// TIA Portal V20 export
DATA_BLOCK "G"   // DB350
{ S7_Optimized_Access := 'TRUE' }
// stored: AutoNumber false, IsRetainMemResEnabled true, MemoryReserve 100, RetainMemoryReserve 100
   VAR RETAIN
      lampTest : Bool;   // lamp test
      settingMode : Bool;   // setting mode active
      jogMode : Bool;   // jog mode active
      scannerReady : Bool;   // scanner ready
      scannerErr : Bool;   // scanner error
      scannerEmpty : Bool;   // scanner empty
      releaseInfeed : Bool;   // release infeed
      auto : Bool;   // automatic mode adjustment
      ack : Bool;   // reset faults general
      ackPC : Bool;   // reset faults pc
      err : Bool;   // fault general
      war : Bool;   // warning general
      info : Bool;   // info general
      pneOk : Bool;   // pneumatic ok
      comOk : Bool;   // communication ok
      "errPs-0F1.1+SGV" : Bool;   // fault voltage monitoring for power supply
      "errAc-0E1+SGV" : Bool;   // fault air conditioner 1 visual
      "errAc-0E2+SGX" : Bool;   // fault air conditioner Xray
      "errAc-0E1.1+SGV" : Bool;   // fault air conditioner 2 visual
      errComPc : Bool;   // fault communication with pc
      errProfinet : Bool;   // fault profinet
      errAdjScanner : Bool;   // fault adjustment scanner
      errAdjTop : Bool;   // fault adjustment top
      errAdjLeft : Bool;   // fault adjustment left
      errAdjRight : Bool;   // fault adjustment right
      errVersion : Bool;   // fault version
      errSafetyModules : Bool;   // fault safety modules
      errNoReleaseInf : Bool;   // fault no release from plc to infeed
      Batch : Struct   // batch info - board data
         stdActive : Bool;   // standardisation batch active
         width : Real;   // board width [mm]
         widthMin : Real;   // board width min [mm]
         widthMax : Real;   // board width max [mm]
         thickness : Real;   // board thickness [mm]
         thicknessMin : Real;   // board thickness min [mm]
         thicknessMax : Real;   // board thickness max [mm]
         widthMeasure : Real;   // board width measured value from sensors [mm]
         thicknessMeasure : Real;   // board thickness measured value from sensor [mm]
         senLeftVal : Real;   // sensor left value [mm]
         senRightVal : Real;   // sensor right value [mm]
         offsetBoard { ExternalWritable := 'False'} : Real;   // offset board to middle [mm] - bigger then zero then board is shifted to the left side
      END_STRUCT;
      Cfg : Struct   // config
         adjScannerActive : Bool;   // adjustment scanner housing active
         adjTopActive : Bool;   // adjustment camera top active
         adjLeftActive : Bool;   // adjustment camera left active
         adjRightActive : Bool;   // adjustment camera right active
         adjTopActiveLinMot : Bool;   // adjustment top active - linear drive
         adjLeftActiveLinMot : Bool;   // adjustment left active - linear drive
         adjRightActiveLinMot : Bool;   // adjustment right active - linear drive
         xrayActive : Bool;   // xray active
         enc1Active : Bool;   // encoder 1 active (infeed)
         senTopActive : Bool;   // sensor top active for random adjustment
         senLeftActive : Bool;   // sensor left active for random adjustment
         senRightActive : Bool;   // sensor right active for random adjustment
         modeBoardPassing : Int;   // 1=left / 2=right / 3=middle
         modeDimension : Int;   // 1=fixed / 2=random width / 3=random thickness / 4=random width + thickness
         modeRandomAdj : Int;   // 1=with sensor / 2=with external data
         enc1Gain : Real;   // encoder 1 gain (infeed)
      END_STRUCT;
      adjScannerOff : Bool;   // adjustment scanner housing off (only manual movement possible )
      adjTopOff : Bool;   // adjustment camera top off (only manual movement possible )
      adjLeftOff : Bool;   // adjustment camera left off (only manual movement possible )
      adjRightOff : Bool;   // adjustment camera right off (only manual movement possible )
   END_VAR
   VAR
      air1Off { ExternalAccessible := 'False'; ExternalVisible := 'False'; ExternalWritable := 'False'} : Bool;
      air2Off { ExternalAccessible := 'False'; ExternalVisible := 'False'; ExternalWritable := 'False'} : Bool;
      airXrayOff { ExternalAccessible := 'False'; ExternalVisible := 'False'; ExternalWritable := 'False'} : Bool;
      airDehOff { ExternalAccessible := 'False'; ExternalVisible := 'False'; ExternalWritable := 'False'} : Bool;
   END_VAR
BEGIN
END_DATA_BLOCK
